PROGRAM F15_AS3_AI
VAR
	
	AI_filter_0: AI_filter;
	AI_filter_1: AI_filter;
	AI_filter_2: AI_filter;
	AI_filter_3: AI_filter;
	AI_filter_4: AI_filter;
	AI_filter_5: AI_filter;
	AI_filter_6: AI_filter;
	AI_filter_7: AI_filter;

END_VAR

VAR PERSISTENT	
	
	Filtertid0 :INT;
	Filtertid1 :INT;
	Filtertid2 :INT;
	Filtertid3 :INT;
	Filtertid4 :INT;
	Filtertid5 :INT;
	Filtertid6 :INT;
	Filtertid7 :INT;
	
	Kalibrering0 :INT;
	Kalibrering1 :INT;
	Kalibrering2 :INT;
	Kalibrering3 :INT;
	Kalibrering4 :INT;
	Kalibrering5 :INT;
	Kalibrering6 :INT;
	Kalibrering7 :INT;
	
END_VAR


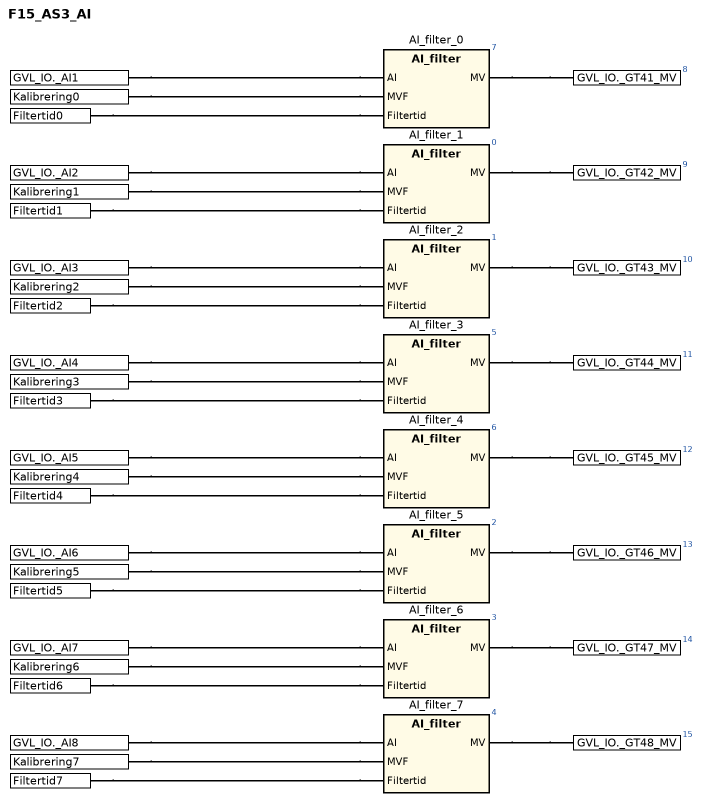
// PAGE
AI_filter_1(AI := GVL_IO._AI2, MVF := Kalibrering1, Filtertid := Filtertid1); // AI_filter
AI_filter_2(AI := GVL_IO._AI3, MVF := Kalibrering2, Filtertid := Filtertid2); // AI_filter
AI_filter_5(AI := GVL_IO._AI6, MVF := Kalibrering5, Filtertid := Filtertid5); // AI_filter
AI_filter_6(AI := GVL_IO._AI7, MVF := Kalibrering6, Filtertid := Filtertid6); // AI_filter
AI_filter_7(AI := GVL_IO._AI8, MVF := Kalibrering7, Filtertid := Filtertid7); // AI_filter
AI_filter_3(AI := GVL_IO._AI4, MVF := Kalibrering3, Filtertid := Filtertid3); // AI_filter
AI_filter_4(AI := GVL_IO._AI5, MVF := Kalibrering4, Filtertid := Filtertid4); // AI_filter
AI_filter_0(AI := GVL_IO._AI1, MVF := Kalibrering0, Filtertid := Filtertid0); // AI_filter
GVL_IO._GT41_MV := AI_filter_0.MV;
GVL_IO._GT42_MV := AI_filter_1.MV;
GVL_IO._GT43_MV := AI_filter_2.MV;
GVL_IO._GT44_MV := AI_filter_3.MV;
GVL_IO._GT45_MV := AI_filter_4.MV;
GVL_IO._GT46_MV := AI_filter_5.MV;
GVL_IO._GT47_MV := AI_filter_6.MV;
GVL_IO._GT48_MV := AI_filter_7.MV;

END_PROGRAM

(* stored: Version 1.1.0.1, ProductVersion 3.1.4020.12
   POU F15_AS3_AI: Id {0e82a025-53df-4dcb-8f90-b5d2a06b7433}, SpecialFunc None *)
